{attribute 'GeneratedUsingTerminal: EL1262-0000-0002'}
{attribute addProperty BoxType "EL1262-0000-0002"}
{attribute addProperty Id "EMPTY_STRUCTURE"}
{attribute addProperty CRC "0"}
{attribute addProperty Size "0"}
TYPE EMPTY_STRUCTURE :
STRUCT
END_STRUCT
END_TYPE
